(* Logix 5000 project; controller DispersionPlc vendor 1 type 14 code 108 rev 34.11; software revision 34.01; part 11 of 22 *)
(* tags used below, declared in another part *)
   AllwaysOff : BOOL;
   block : BOOL;
   Dn_DataMap_In : INT[12];
   Dn_DataMap_out : INT[12];
   InputIdx : DINT;
   ONS : BOOL[32];
   OutPutIdx : DINT;
   ReffBit : BOOL;
   Temp : BOOL;
   TurningOnReffBit : BOOL;
   VfdReff : VFD;
   _JISdebug : DINT;
   AFB : BOOL;
   AFI : BOOL;
   Bulk_Tank_T52_Level_Lamp : ALIAS FOR Local:1:O.Data[12].3;
   Bulk_Tank_T53_Level_Lamp : ALIAS FOR Local:1:O.Data[12].4;
   DispersionAlarms : BOOL[256];
   FE_4303 : REAL;
   FE_4303_Out : REAL;
   FE_4303_STORAGE : REAL[1000];
   FE_4303_WEIGHT : REAL[100];
   MCR_Bulk : ALIAS FOR Local:1:I.Data[33].4;
   Micro_Motion : COUNTER;
   micromotion : TIMER;
   MICROMOTION_POUNDS : REAL;
   MICROMOTION_PULSE_COUNT_COUNT_INPUT : ALIAS FOR Local:1:I.Data[32].1;
   MICROMOTION_SF : REAL;
   MIRCOMOITION_ENABLE : ALIAS FOR Local:1:I.Data[32].7;
   MM_Gal_Ach : ALIAS FOR Local:1:I.Data[32].2;
   MMI_Mixer_T52_RUN_PB : BOOL;
   MMI_Mixer_T53_RUN_PB : BOOL;
   MMI_T52_Level : INT;
   MMI_T52_WARN_BYPASS : BOOL;
   MMI_T53_Level : INT;
   MMI_T53_WARN_BYPASS : BOOL;
   MMI_XV_5201_PB : BOOL;
   MMI_XV_5202_PB : BOOL;
   MMI_XV_5301_PB : BOOL;
   MMI_XV_5302_PB : BOOL;
   NM_4303_O2_SIGNAL : REAL;
   NM_4303_SIGNAL_AVERAGE_STORAGE : REAL[1000];
   NM_4303_SIGNAL_AVERAGE_WEIGHT : REAL[100];
   RG_T52 : REAL;
   RG_T52_AI_Holding : REAL;
   RG_T52_AI_Raw : INT;
   RG_T52_AI_Samples : DINT;
   RG_T52_Holding1 : REAL;
   RG_T52_Min_Tank_Value : INT;
   RG_T52_OffSet : REAL;
   RG_T52_REMAINDER : REAL;
   RG_T52_Sf : REAL;
   RG_T53 : REAL;
   RG_T53_AI_Holding : REAL;
   RG_T53_AI_Raw : INT;
   RG_T53_AI_Samples : DINT;
   RG_T53_Holding1 : REAL;
   RG_T53_Min_Tank_Value : INT;
   RG_T53_OffSet : REAL;
   RG_T53_REMAINDER : REAL;
   RG_T53_Sf : REAL;
   SP : REAL;
   T52_Mixer : VFD;
   T52_Mixer_STOP : TIMER;
   T52_Ons : BOOL[32];
   T52_Selected_For_Pumping : BOOL;
   T52_Tank_Max_Lbs : REAL;
   T52_WARN_BYPASS : BOOL;
   T53_Mixer : VFD;
   T53_Mixer_STOP : TIMER;
   T53_Ons : BOOL[32];
   T53_Selected_For_Pumping : BOOL;
   T53_Tank_Max_Lbs : REAL;
   T53_WARN_BYPASS : BOOL;
   TOGGLE : BOOL;
   Trans_Pump_P52_Aux : ALIAS FOR Local:1:I.Data[33].0;
   Trans_Pump_P53_Aux : ALIAS FOR Local:1:I.Data[33].1;
   Trans_Pump_T52_Run : ALIAS FOR Local:1:O.Data[13].1;
   Trans_Pump_T52_Run_Lamp : ALIAS FOR Local:1:O.Data[12].0;
   Trans_Pump_T52_Run_PB : ALIAS FOR Local:1:I.Data[27].0;
   Trans_Pump_T52_Stop_PB : ALIAS FOR Local:1:I.Data[27].1;
   Trans_Pump_T53_Run : ALIAS FOR Local:1:O.Data[13].2;
   Trans_Pump_T53_Run_Lamp : ALIAS FOR Local:1:O.Data[12].1;
   Trans_Pump_T53_Run_PB : ALIAS FOR Local:1:I.Data[27].2;
   Trans_Pump_T53_Stop_PB : ALIAS FOR Local:1:I.Data[27].3;
   XV_5201 : ALIAS FOR Local:1:O.Data[12].8;
   XV_5202 : ALIAS FOR Local:1:O.Data[12].9;
   XV_5301 : ALIAS FOR Local:1:O.Data[12].6;
   XV_5302 : ALIAS FOR Local:1:O.Data[12].7;
(* MainProgram, continued *)

ROUTINE T52   (* ladder *)
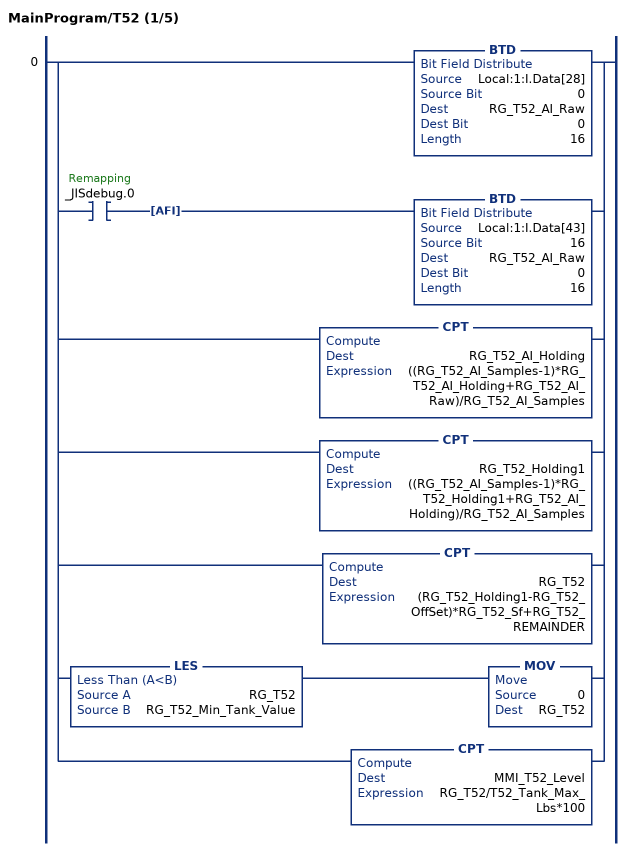
   0: [BTD(Local:1:I.Data[28],0,RG_T52_AI_Raw,0,16) ,XIC(_JISdebug.0) AFI() BTD(Local:1:I.Data[43],16,RG_T52_AI_Raw,0,16) ,CPT(RG_T52_AI_Holding,((RG_T52_AI_Samples-1)*RG_T52_AI_Holding+RG_T52_AI_Raw)/RG_T52_AI_Samples) ,CPT(RG_T52_Holding1,((RG_T52_AI_Samples-1)*RG_T52_Holding1+RG_T52_AI_Holding)/RG_T52_AI_Samples) ,CPT(RG_T52,(RG_T52_Holding1-RG_T52_OffSet)*RG_T52_Sf+RG_T52_REMAINDER) ,LES(RG_T52,RG_T52_Min_Tank_Value) MOV(0,RG_T52) ,CPT(MMI_T52_Level,RG_T52/T52_Tank_Max_Lbs*100) ];
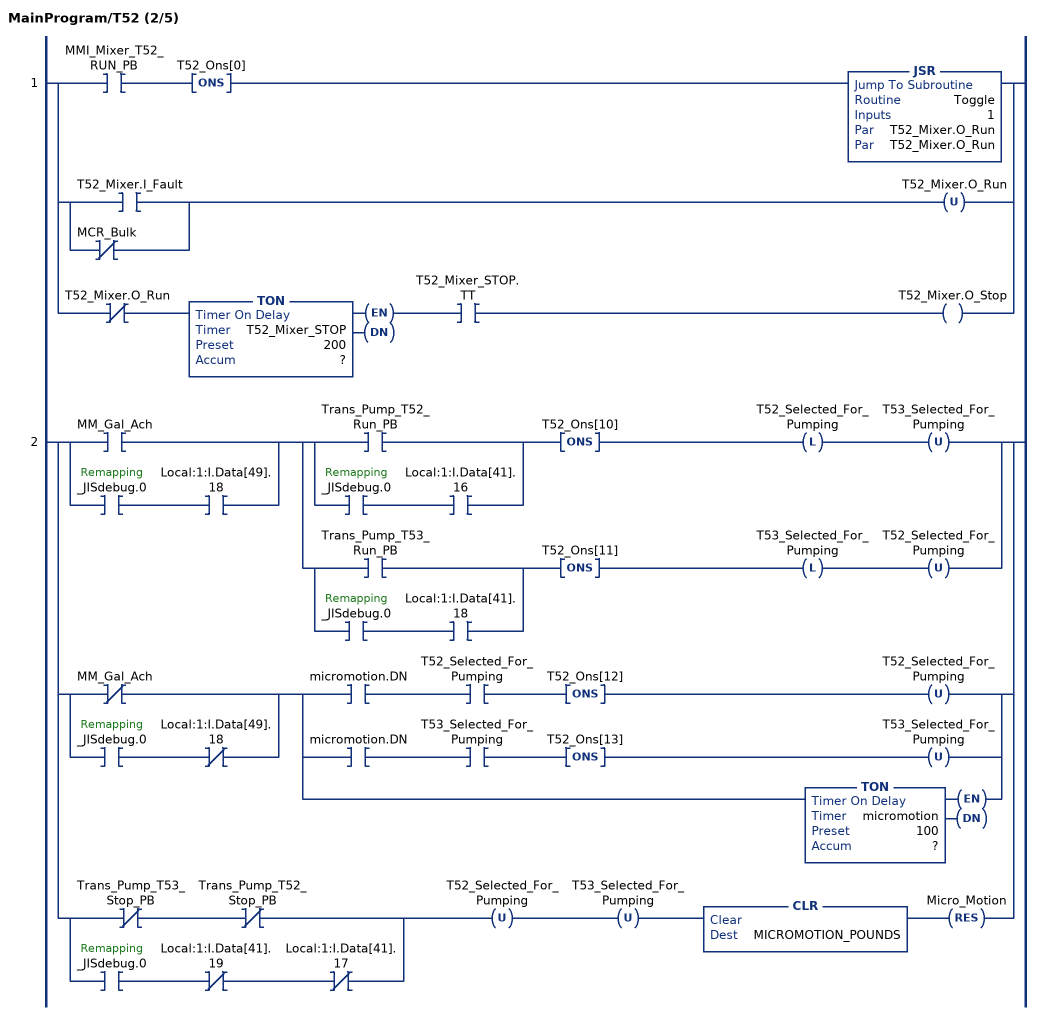
   1: [XIC(MMI_Mixer_T52_RUN_PB) ONS(T52_Ons[0]) JSR(Toggle,1,T52_Mixer.O_Run,T52_Mixer.O_Run) ,[XIC(T52_Mixer.I_Fault) ,XIO(MCR_Bulk) ] OTU(T52_Mixer.O_Run) ,XIO(T52_Mixer.O_Run) TON(T52_Mixer_STOP,?,?) XIC(T52_Mixer_STOP.TT) OTE(T52_Mixer.O_Stop) ];
   2: [[XIC(MM_Gal_Ach) ,XIC(_JISdebug.0) XIC(Local:1:I.Data[49].18) ] [[XIC(Trans_Pump_T52_Run_PB) ,XIC(_JISdebug.0) XIC(Local:1:I.Data[41].16) ] ONS(T52_Ons[10]) OTL(T52_Selected_For_Pumping) OTU(T53_Selected_For_Pumping) ,[XIC(Trans_Pump_T53_Run_PB) ,XIC(_JISdebug.0) XIC(Local:1:I.Data[41].18) ] ONS(T52_Ons[11]) OTL(T53_Selected_For_Pumping) OTU(T52_Selected_For_Pumping) ] ,[XIO(MM_Gal_Ach) ,XIC(_JISdebug.0) XIO(Local:1:I.Data[49].18) ] [XIC(micromotion.DN) XIC(T52_Selected_For_Pumping) ONS(T52_Ons[12]) OTU(T52_Selected_For_Pumping) ,XIC(micromotion.DN) XIC(T53_Selected_For_Pumping) ONS(T52_Ons[13]) OTU(T53_Selected_For_Pumping) ,TON(micromotion,?,?) ] ,[XIO(Trans_Pump_T53_Stop_PB) XIO(Trans_Pump_T52_Stop_PB) ,XIC(_JISdebug.0) XIO(Local:1:I.Data[41].19) XIO(Local:1:I.Data[41].17) ] OTU(T52_Selected_For_Pumping) OTU(T53_Selected_For_Pumping) CLR(MICROMOTION_POUNDS) RES(Micro_Motion) ];
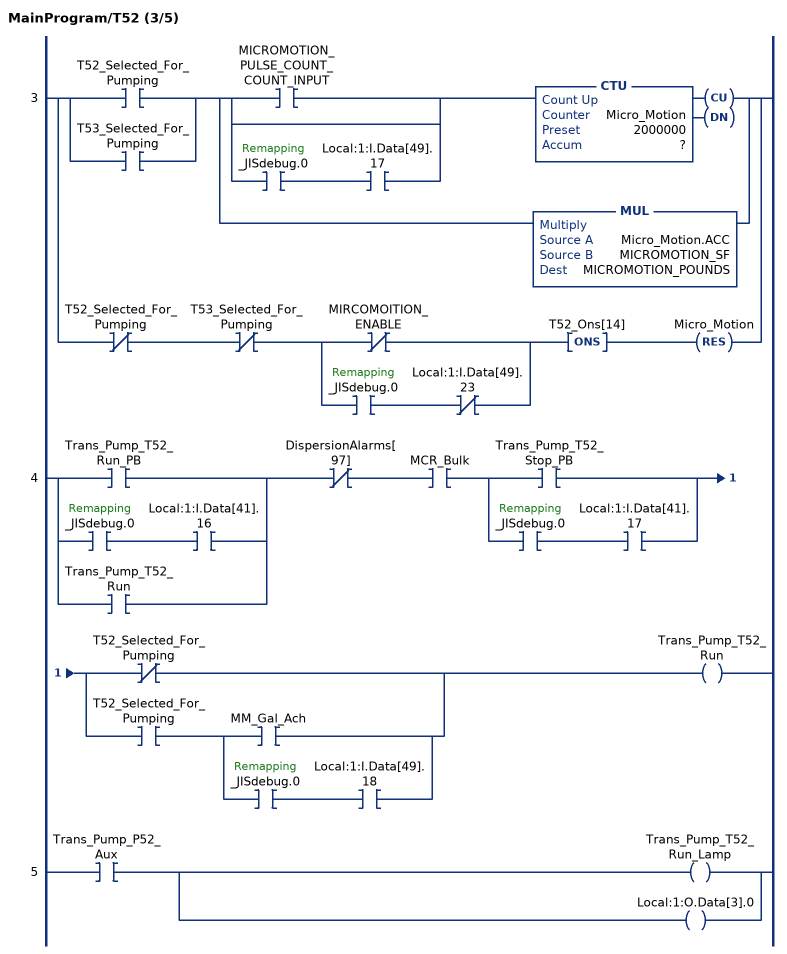
   3: [[XIC(T52_Selected_For_Pumping) ,XIC(T53_Selected_For_Pumping) ] [[XIC(MICROMOTION_PULSE_COUNT_COUNT_INPUT) ,,XIC(_JISdebug.0) XIC(Local:1:I.Data[49].17) ] CTU(Micro_Motion,?,?) ,MUL(Micro_Motion.ACC,MICROMOTION_SF,MICROMOTION_POUNDS) ] ,XIO(T52_Selected_For_Pumping) XIO(T53_Selected_For_Pumping) [XIO(MIRCOMOITION_ENABLE) ,XIC(_JISdebug.0) XIO(Local:1:I.Data[49].23) ] ONS(T52_Ons[14]) RES(Micro_Motion) ];
   4: [XIC(Trans_Pump_T52_Run_PB) ,XIC(_JISdebug.0) XIC(Local:1:I.Data[41].16) ,XIC(Trans_Pump_T52_Run) ]XIO(DispersionAlarms[97])XIC(MCR_Bulk)[XIC(Trans_Pump_T52_Stop_PB) ,XIC(_JISdebug.0) XIC(Local:1:I.Data[41].17) ][XIO(T52_Selected_For_Pumping) ,XIC(T52_Selected_For_Pumping) [XIC(MM_Gal_Ach) ,XIC(_JISdebug.0) XIC(Local:1:I.Data[49].18) ] ]OTE(Trans_Pump_T52_Run);
   5: XIC(Trans_Pump_P52_Aux)[OTE(Trans_Pump_T52_Run_Lamp) ,OTE(Local:1:O.Data[3].0) ];
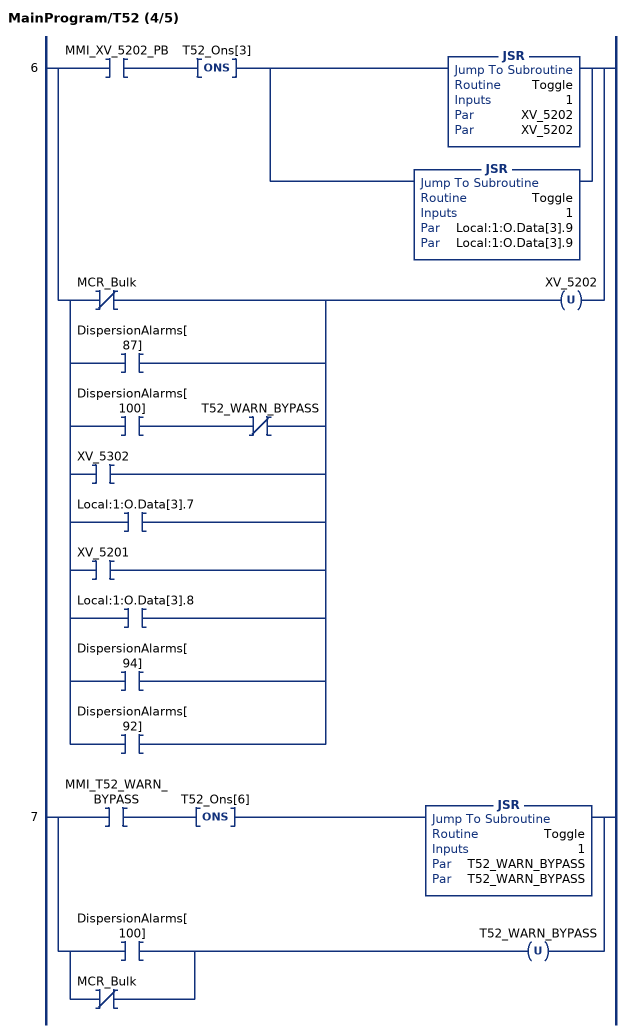
   6: [XIC(MMI_XV_5202_PB) ONS(T52_Ons[3]) [JSR(Toggle,1,XV_5202,XV_5202) ,JSR(Toggle,1,Local:1:O.Data[3].9,Local:1:O.Data[3].9) ] ,[XIO(MCR_Bulk) ,XIC(DispersionAlarms[87]) ,XIC(DispersionAlarms[100]) XIO(T52_WARN_BYPASS) ,XIC(XV_5302) ,XIC(Local:1:O.Data[3].7) ,XIC(XV_5201) ,XIC(Local:1:O.Data[3].8) ,XIC(DispersionAlarms[94]) ,XIC(DispersionAlarms[92]) ] OTU(XV_5202) ];
   7: [XIC(MMI_T52_WARN_BYPASS) ONS(T52_Ons[6]) JSR(Toggle,1,T52_WARN_BYPASS,T52_WARN_BYPASS) ,[XIC(DispersionAlarms[100]) ,XIO(MCR_Bulk) ] OTU(T52_WARN_BYPASS) ];
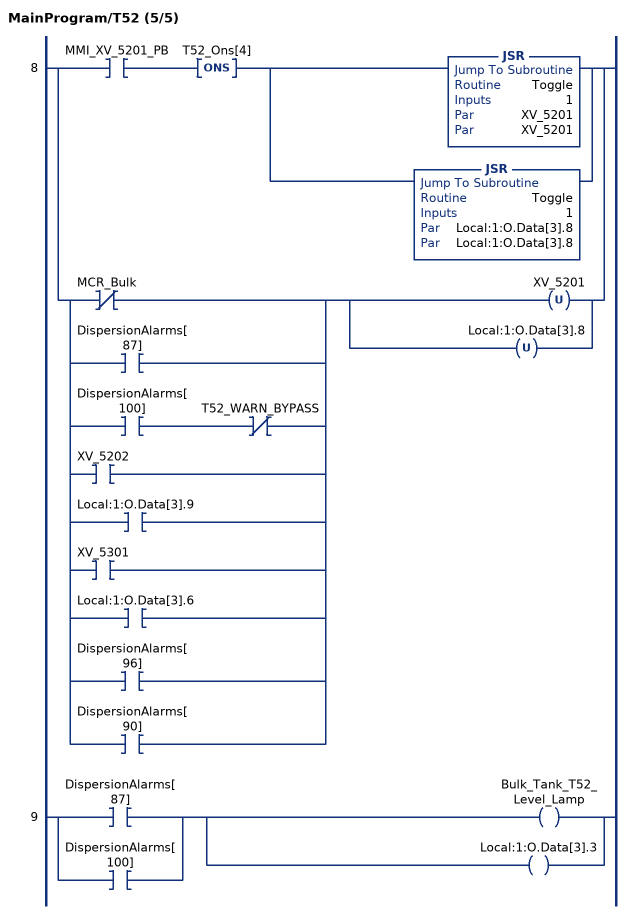
   8: [XIC(MMI_XV_5201_PB) ONS(T52_Ons[4]) [JSR(Toggle,1,XV_5201,XV_5201) ,JSR(Toggle,1,Local:1:O.Data[3].8,Local:1:O.Data[3].8) ] ,[XIO(MCR_Bulk) ,XIC(DispersionAlarms[87]) ,XIC(DispersionAlarms[100]) XIO(T52_WARN_BYPASS) ,XIC(XV_5202) ,XIC(Local:1:O.Data[3].9) ,XIC(XV_5301) ,XIC(Local:1:O.Data[3].6) ,XIC(DispersionAlarms[96]) ,XIC(DispersionAlarms[90]) ] [OTU(XV_5201) ,OTU(Local:1:O.Data[3].8) ] ];
   9: [XIC(DispersionAlarms[87]) ,XIC(DispersionAlarms[100]) ][OTE(Bulk_Tank_T52_Level_Lamp) ,OTE(Local:1:O.Data[3].3) ];
END_ROUTINE

ROUTINE T53   (* ladder *)
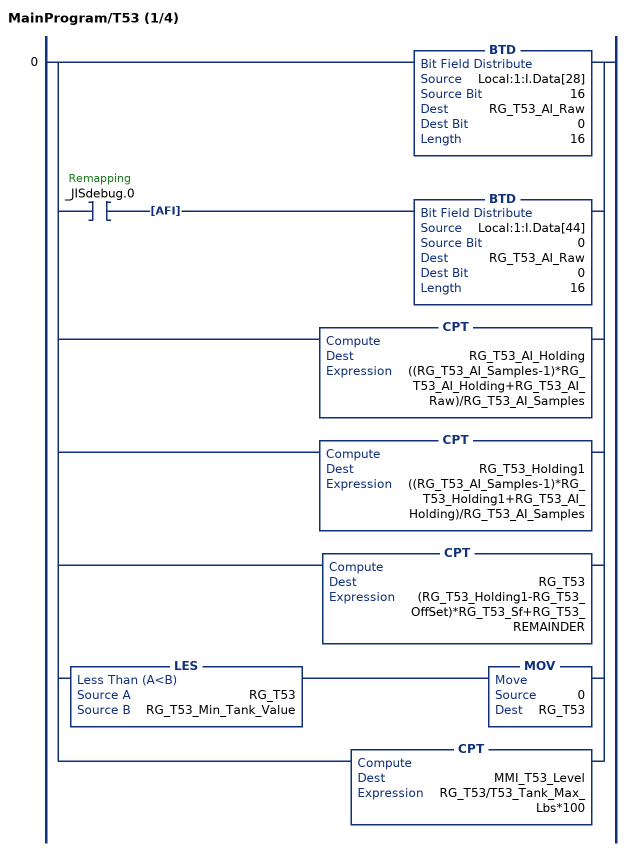
   0: [BTD(Local:1:I.Data[28],16,RG_T53_AI_Raw,0,16) ,XIC(_JISdebug.0) AFI() BTD(Local:1:I.Data[44],0,RG_T53_AI_Raw,0,16) ,CPT(RG_T53_AI_Holding,((RG_T53_AI_Samples-1)*RG_T53_AI_Holding+RG_T53_AI_Raw)/RG_T53_AI_Samples) ,CPT(RG_T53_Holding1,((RG_T53_AI_Samples-1)*RG_T53_Holding1+RG_T53_AI_Holding)/RG_T53_AI_Samples) ,CPT(RG_T53,(RG_T53_Holding1-RG_T53_OffSet)*RG_T53_Sf+RG_T53_REMAINDER) ,LES(RG_T53,RG_T53_Min_Tank_Value) MOV(0,RG_T53) ,CPT(MMI_T53_Level,RG_T53/T53_Tank_Max_Lbs*100) ];
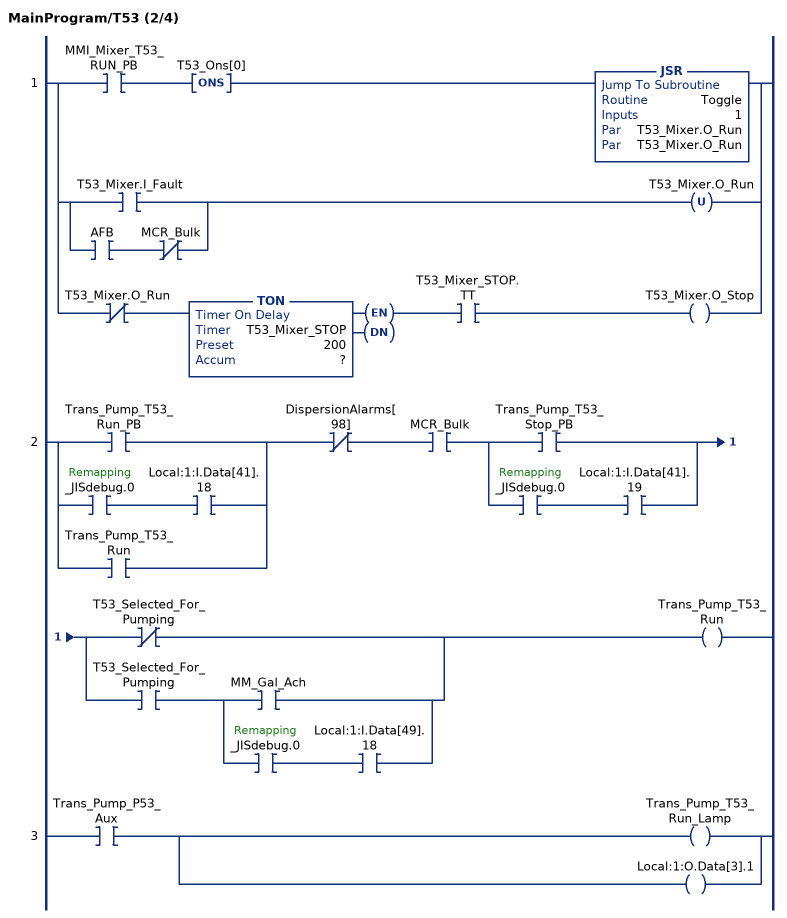
   1: [XIC(MMI_Mixer_T53_RUN_PB) ONS(T53_Ons[0]) JSR(Toggle,1,T53_Mixer.O_Run,T53_Mixer.O_Run) ,[XIC(T53_Mixer.I_Fault) ,XIC(AFB) XIO(MCR_Bulk) ] OTU(T53_Mixer.O_Run) ,XIO(T53_Mixer.O_Run) TON(T53_Mixer_STOP,?,?) XIC(T53_Mixer_STOP.TT) OTE(T53_Mixer.O_Stop) ];
   2: [XIC(Trans_Pump_T53_Run_PB) ,XIC(_JISdebug.0) XIC(Local:1:I.Data[41].18) ,XIC(Trans_Pump_T53_Run) ]XIO(DispersionAlarms[98])XIC(MCR_Bulk)[XIC(Trans_Pump_T53_Stop_PB) ,XIC(_JISdebug.0) XIC(Local:1:I.Data[41].19) ][XIO(T53_Selected_For_Pumping) ,XIC(T53_Selected_For_Pumping) [XIC(MM_Gal_Ach) ,XIC(_JISdebug.0) XIC(Local:1:I.Data[49].18) ] ]OTE(Trans_Pump_T53_Run);
   3: XIC(Trans_Pump_P53_Aux)[OTE(Trans_Pump_T53_Run_Lamp) ,OTE(Local:1:O.Data[3].1) ];
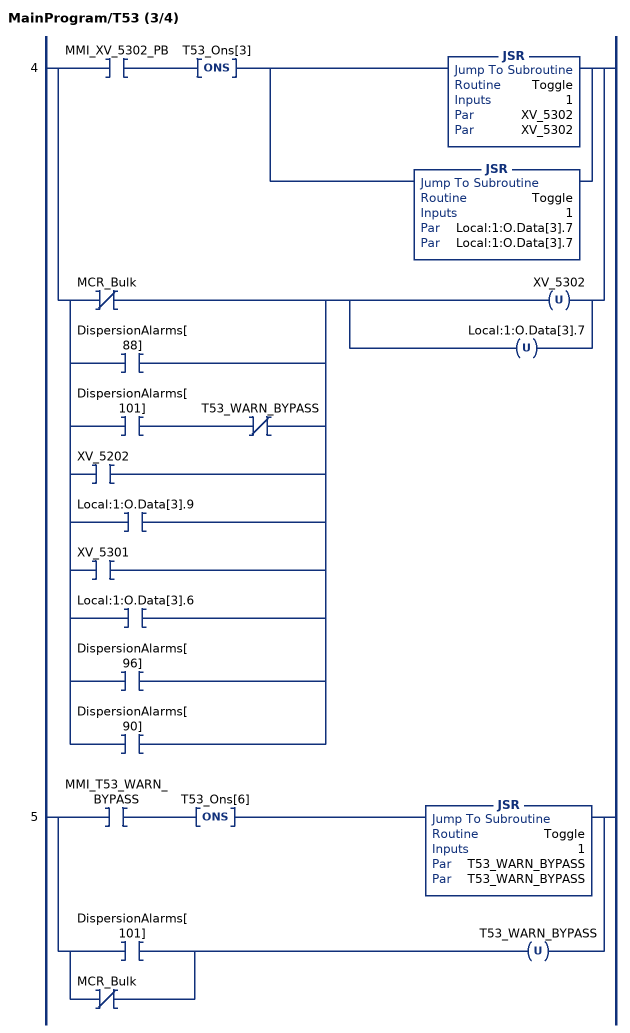
   4: [XIC(MMI_XV_5302_PB) ONS(T53_Ons[3]) [JSR(Toggle,1,XV_5302,XV_5302) ,JSR(Toggle,1,Local:1:O.Data[3].7,Local:1:O.Data[3].7) ] ,[XIO(MCR_Bulk) ,XIC(DispersionAlarms[88]) ,XIC(DispersionAlarms[101]) XIO(T53_WARN_BYPASS) ,XIC(XV_5202) ,XIC(Local:1:O.Data[3].9) ,XIC(XV_5301) ,XIC(Local:1:O.Data[3].6) ,XIC(DispersionAlarms[96]) ,XIC(DispersionAlarms[90]) ] [OTU(XV_5302) ,OTU(Local:1:O.Data[3].7) ] ];
   5: [XIC(MMI_T53_WARN_BYPASS) ONS(T53_Ons[6]) JSR(Toggle,1,T53_WARN_BYPASS,T53_WARN_BYPASS) ,[XIC(DispersionAlarms[101]) ,XIO(MCR_Bulk) ] OTU(T53_WARN_BYPASS) ];
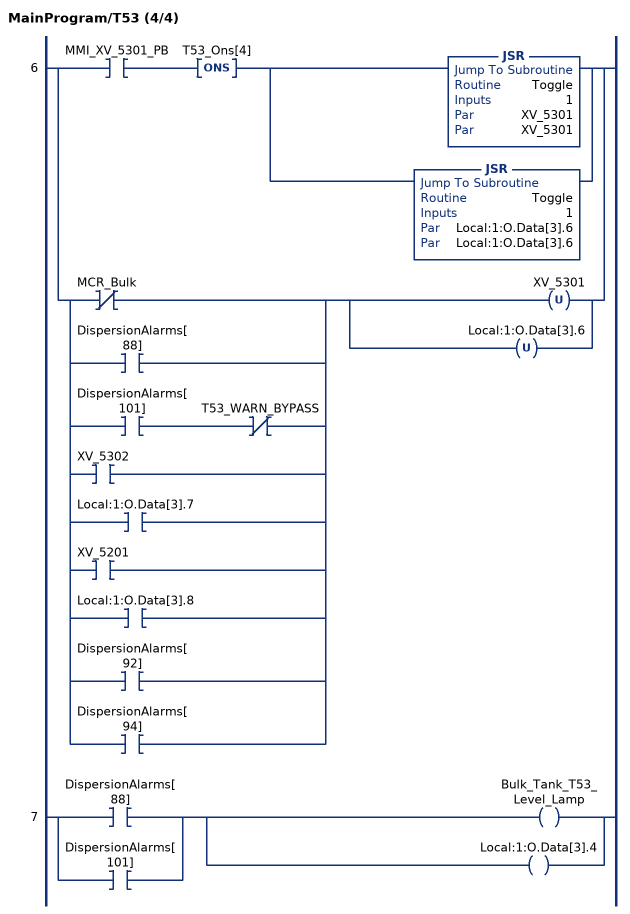
   6: [XIC(MMI_XV_5301_PB) ONS(T53_Ons[4]) [JSR(Toggle,1,XV_5301,XV_5301) ,JSR(Toggle,1,Local:1:O.Data[3].6,Local:1:O.Data[3].6) ] ,[XIO(MCR_Bulk) ,XIC(DispersionAlarms[88]) ,XIC(DispersionAlarms[101]) XIO(T53_WARN_BYPASS) ,XIC(XV_5302) ,XIC(Local:1:O.Data[3].7) ,XIC(XV_5201) ,XIC(Local:1:O.Data[3].8) ,XIC(DispersionAlarms[92]) ,XIC(DispersionAlarms[94]) ] [OTU(XV_5301) ,OTU(Local:1:O.Data[3].6) ] ];
   7: [XIC(DispersionAlarms[88]) ,XIC(DispersionAlarms[101]) ][OTE(Bulk_Tank_T53_Level_Lamp) ,OTE(Local:1:O.Data[3].4) ];
END_ROUTINE

ROUTINE Toggle   (* ladder *)
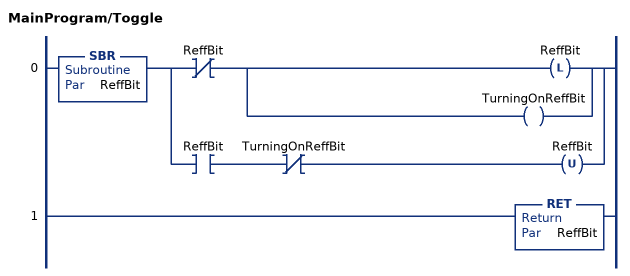
   0: SBR(ReffBit)[XIO(ReffBit) [OTL(ReffBit) ,OTE(TurningOnReffBit) ] ,XIC(ReffBit) XIO(TurningOnReffBit) OTU(ReffBit) ];
   1: RET(ReffBit);
END_ROUTINE

ROUTINE Vfd_Interface   (* ladder *)
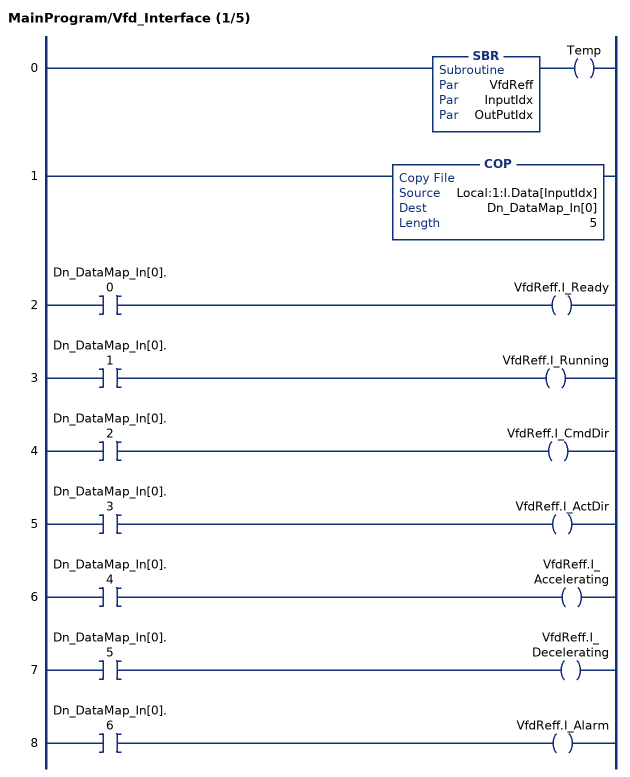
   0: SBR(VfdReff,InputIdx,OutPutIdx)OTE(Temp);
   1: COP(Local:1:I.Data[InputIdx],Dn_DataMap_In[0],5);
   2: XIC(Dn_DataMap_In[0].0)OTE(VfdReff.I_Ready);
   3: XIC(Dn_DataMap_In[0].1)OTE(VfdReff.I_Running);
   4: XIC(Dn_DataMap_In[0].2)OTE(VfdReff.I_CmdDir);
   5: XIC(Dn_DataMap_In[0].3)OTE(VfdReff.I_ActDir);
   6: XIC(Dn_DataMap_In[0].4)OTE(VfdReff.I_Accelerating);
   7: XIC(Dn_DataMap_In[0].5)OTE(VfdReff.I_Decelerating);
   8: XIC(Dn_DataMap_In[0].6)OTE(VfdReff.I_Alarm);
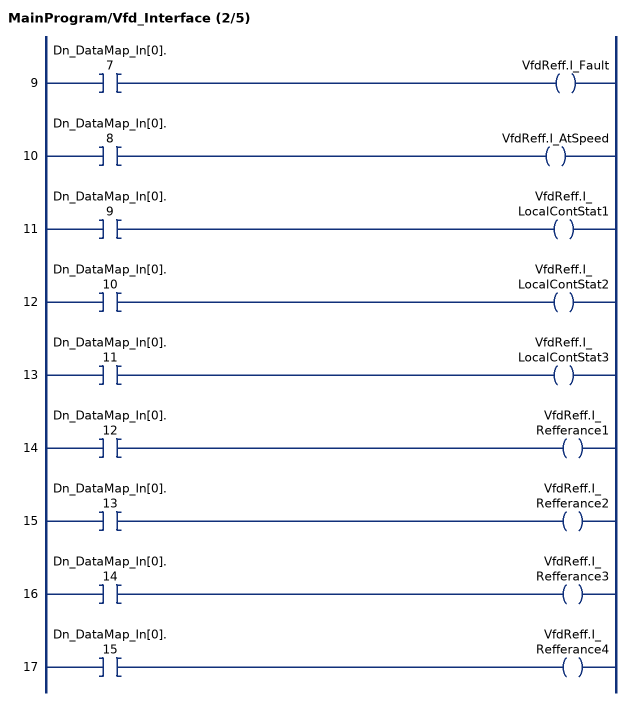
   9: XIC(Dn_DataMap_In[0].7)OTE(VfdReff.I_Fault);
   10: XIC(Dn_DataMap_In[0].8)OTE(VfdReff.I_AtSpeed);
   11: XIC(Dn_DataMap_In[0].9)OTE(VfdReff.I_LocalContStat1);
   12: XIC(Dn_DataMap_In[0].10)OTE(VfdReff.I_LocalContStat2);
   13: XIC(Dn_DataMap_In[0].11)OTE(VfdReff.I_LocalContStat3);
   14: XIC(Dn_DataMap_In[0].12)OTE(VfdReff.I_Refferance1);
   15: XIC(Dn_DataMap_In[0].13)OTE(VfdReff.I_Refferance2);
   16: XIC(Dn_DataMap_In[0].14)OTE(VfdReff.I_Refferance3);
   17: XIC(Dn_DataMap_In[0].15)OTE(VfdReff.I_Refferance4);
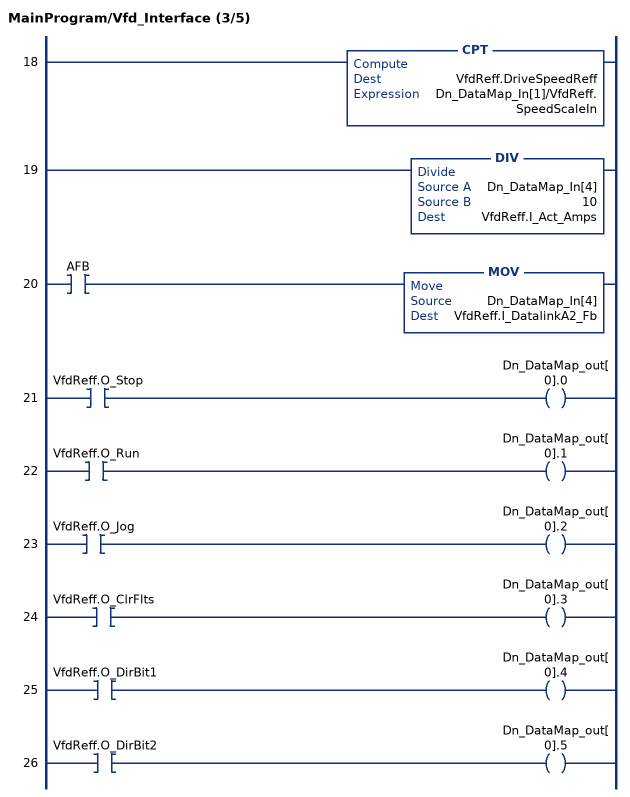
   18: CPT(VfdReff.DriveSpeedReff,Dn_DataMap_In[1]/VfdReff.SpeedScaleIn);
   19: DIV(Dn_DataMap_In[4],10,VfdReff.I_Act_Amps);
   20: XIC(AFB)MOV(Dn_DataMap_In[4],VfdReff.I_DatalinkA2_Fb);
   21: XIC(VfdReff.O_Stop)OTE(Dn_DataMap_out[0].0);
   22: XIC(VfdReff.O_Run)OTE(Dn_DataMap_out[0].1);
   23: XIC(VfdReff.O_Jog)OTE(Dn_DataMap_out[0].2);
   24: XIC(VfdReff.O_ClrFlts)OTE(Dn_DataMap_out[0].3);
   25: XIC(VfdReff.O_DirBit1)OTE(Dn_DataMap_out[0].4);
   26: XIC(VfdReff.O_DirBit2)OTE(Dn_DataMap_out[0].5);
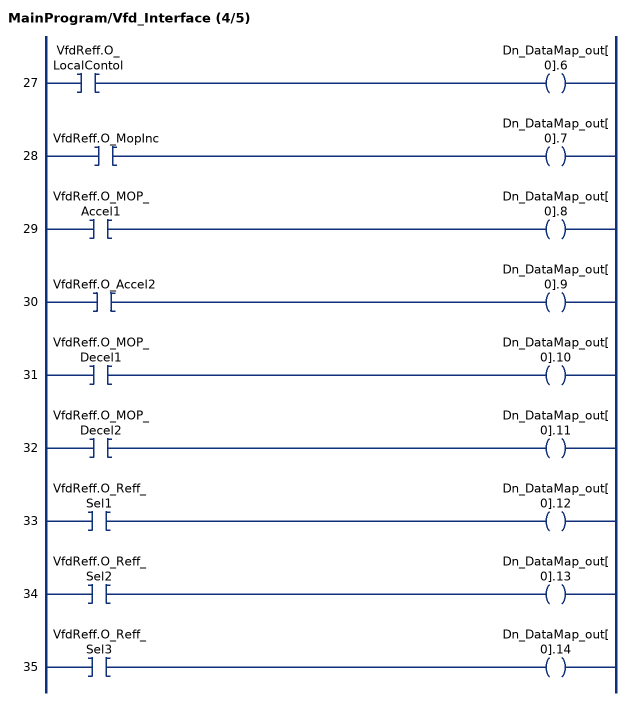
   27: XIC(VfdReff.O_LocalContol)OTE(Dn_DataMap_out[0].6);
   28: XIC(VfdReff.O_MopInc)OTE(Dn_DataMap_out[0].7);
   29: XIC(VfdReff.O_MOP_Accel1)OTE(Dn_DataMap_out[0].8);
   30: XIC(VfdReff.O_Accel2)OTE(Dn_DataMap_out[0].9);
   31: XIC(VfdReff.O_MOP_Decel1)OTE(Dn_DataMap_out[0].10);
   32: XIC(VfdReff.O_MOP_Decel2)OTE(Dn_DataMap_out[0].11);
   33: XIC(VfdReff.O_Reff_Sel1)OTE(Dn_DataMap_out[0].12);
   34: XIC(VfdReff.O_Reff_Sel2)OTE(Dn_DataMap_out[0].13);
   35: XIC(VfdReff.O_Reff_Sel3)OTE(Dn_DataMap_out[0].14);
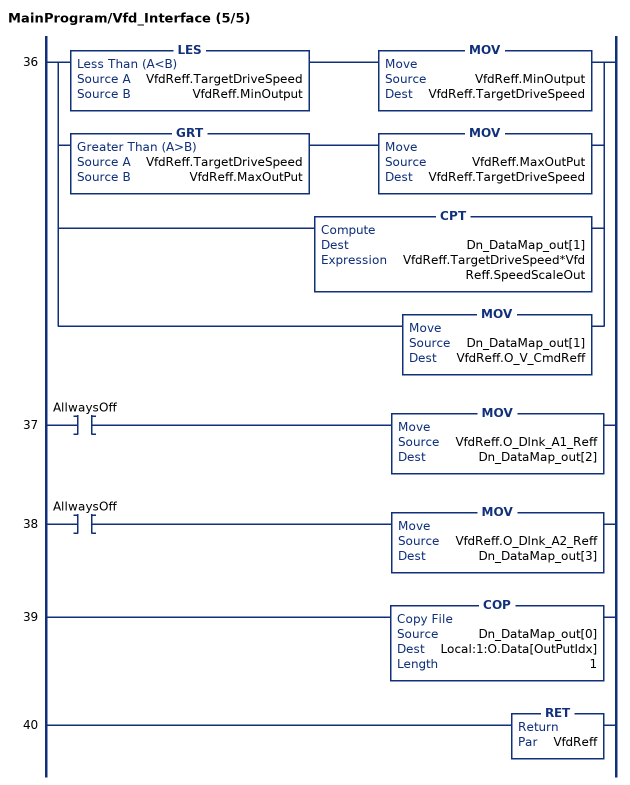
   36: [LES(VfdReff.TargetDriveSpeed,VfdReff.MinOutput) MOV(VfdReff.MinOutput,VfdReff.TargetDriveSpeed) ,GRT(VfdReff.TargetDriveSpeed,VfdReff.MaxOutPut) MOV(VfdReff.MaxOutPut,VfdReff.TargetDriveSpeed) ,CPT(Dn_DataMap_out[1],VfdReff.TargetDriveSpeed*VfdReff.SpeedScaleOut) ,MOV(Dn_DataMap_out[1],VfdReff.O_V_CmdReff) ];
   37: XIC(AllwaysOff)MOV(VfdReff.O_Dlnk_A1_Reff,Dn_DataMap_out[2]);
   38: XIC(AllwaysOff)MOV(VfdReff.O_Dlnk_A2_Reff,Dn_DataMap_out[3]);
   39: COP(Dn_DataMap_out[0],Local:1:O.Data[OutPutIdx],1);
   40: RET(VfdReff);
END_ROUTINE
END_PROGRAM

PROGRAM PIDLoops   (* main routine Main *)
VAR
   BNOT_01 : FBD_BOOLEAN_NOT := (Out := 1);
   MAVE_01 : MOVING_AVERAGE := (SampleEnable := 1, NumberOfSamples := 1);
   MAVE_02 : MOVING_AVERAGE := (SampleEnable := 1, NumberOfSamples := 1);
   PIDE_01 : PID_ENHANCED := (PVEUMax := 100.0, SPHLimit := 100.0, RatioProg := 1.0, RatioOper := 1.0, RatioHLimit := 1.0, RatioLLimit := 1.0, CVEUMax := 100.0, CVHLimit := 100.0, PVEDerivative := 1, RTSTime := 1);
   SEL_01 : SELECT;
END_VAR

ROUTINE Main   (* ladder *)
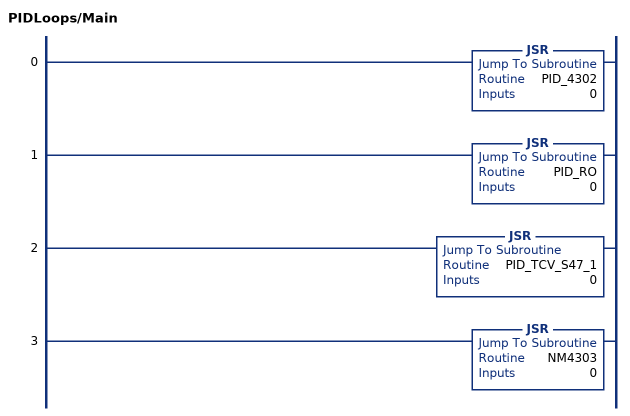
   0: JSR(PID_4302,0);
   1: JSR(PID_RO,0);
   2: JSR(PID_TCV_S47_1,0);
   3: JSR(NM4303,0);
END_ROUTINE

ROUTINE NM4303   (* function block diagram *)
   SHEET 1
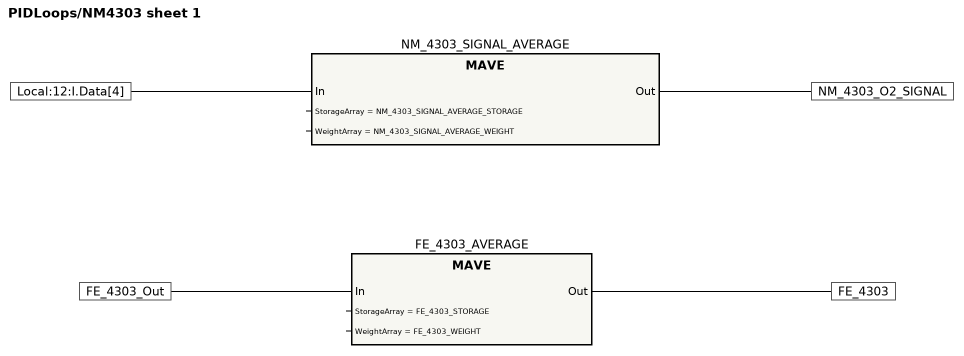
   NM_4303_SIGNAL_AVERAGE : MAVE(In := Local:12:I.Data[4], StorageArray := NM_4303_SIGNAL_AVERAGE_STORAGE, WeightArray := NM_4303_SIGNAL_AVERAGE_WEIGHT);
   FE_4303_AVERAGE : MAVE(In := FE_4303_Out, StorageArray := FE_4303_STORAGE, WeightArray := FE_4303_WEIGHT);
   NM_4303_O2_SIGNAL := NM_4303_SIGNAL_AVERAGE.Out;
   FE_4303 := FE_4303_AVERAGE.Out;
END_ROUTINE

ROUTINE PID_4302   (* function block diagram *)
   SHEET 1
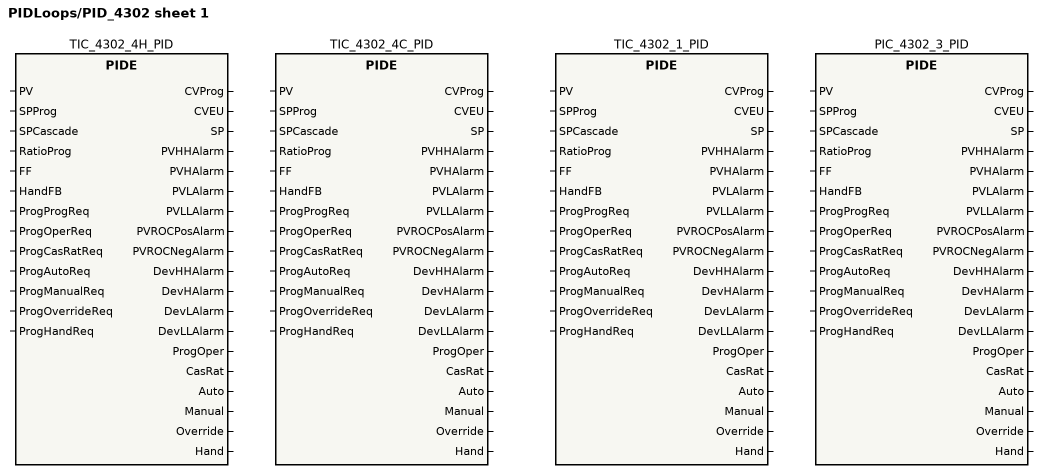
   TIC_4302_4H_PID : PIDE();   // unwired pins: PV SPProg SPCascade RatioProg CVProg FF HandFB ProgProgReq ProgOperReq ProgCasRatReq ProgAutoReq ProgManualReq ProgOverrideReq ProgHandReq CVEU SP PVHHAlarm PVHAlarm PVLAlarm PVLLAlarm PVROCPosAlarm PVROCNegAlarm DevHHAlarm DevHAlarm DevLAlarm DevLLAlarm ProgOper CasRat Auto Manual Override Hand
   TIC_4302_4C_PID : PIDE();   // unwired pins: PV SPProg SPCascade RatioProg CVProg FF HandFB ProgProgReq ProgOperReq ProgCasRatReq ProgAutoReq ProgManualReq ProgOverrideReq ProgHandReq CVEU SP PVHHAlarm PVHAlarm PVLAlarm PVLLAlarm PVROCPosAlarm PVROCNegAlarm DevHHAlarm DevHAlarm DevLAlarm DevLLAlarm ProgOper CasRat Auto Manual Override Hand
   TIC_4302_1_PID : PIDE();   // unwired pins: PV SPProg SPCascade RatioProg CVProg FF HandFB ProgProgReq ProgOperReq ProgCasRatReq ProgAutoReq ProgManualReq ProgOverrideReq ProgHandReq CVEU SP PVHHAlarm PVHAlarm PVLAlarm PVLLAlarm PVROCPosAlarm PVROCNegAlarm DevHHAlarm DevHAlarm DevLAlarm DevLLAlarm ProgOper CasRat Auto Manual Override Hand
   PIC_4302_3_PID : PIDE();   // unwired pins: PV SPProg SPCascade RatioProg CVProg FF HandFB ProgProgReq ProgOperReq ProgCasRatReq ProgAutoReq ProgManualReq ProgOverrideReq ProgHandReq CVEU SP PVHHAlarm PVHAlarm PVLAlarm PVLLAlarm PVROCPosAlarm PVROCNegAlarm DevHHAlarm DevHAlarm DevLAlarm DevLLAlarm ProgOper CasRat Auto Manual Override Hand
END_ROUTINE
